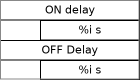
VISUALIZATION UI_Time  // 140x80
VAR_IN_OUT
	settings : Room_Settings_TimeSettings;
END_VAR
    Rectangle (40,60 100x20), "%i s", text variable: settings.nOn
        OnMouseClick: write the text variable via Default
    Rectangle (0,40 140x20), "OFF Delay"
    Rectangle (0,0 140x20), "ON delay"
    Rectangle (40,20 100x20), "%i s", text variable: settings.nOff
        OnMouseClick: write the text variable via Default
END_VISUALIZATION

(* stored: Version 1.1.0.1
   Visu UI_Time: Id {c5fad084-02c2-40ed-a415-b87b6faec236} *)
